// TIA Portal V19 export
TYPE "lexchangetray_typeUnEmn_toHandlingXyzReq"
// Type: Bool
// stored: Access Published
   STRUCT
      transferEnable : Bool;   // Manual mode parameters for axis control interface
   END_STRUCT;
END_TYPE
